{attribute 'qualified_only'}
VAR_GLOBAL CONSTANT
  MaxDevicesSearchCount : UINT := 200;
  MaxDeviceToBeFound : UINT := 10;
  MaxSlavesToBeFound : UINT := 200;
END_VAR

(* stored: Version 1.1.0.1
   GVL Parameter: Id {45938ee2-c814-47c6-928c-f40125e2ba09}, ParameterList True *)
